FUNCTION_BLOCK Test_TimestampAsFilenameString EXTENDS TUnitTestBase
VAR
END_VAR

METHOD  Execute
VAR_INST
    TimeStruct : TIMESTRUCT := (wDay := 23, wMonth := 12, wYear := 1945, wHour := 22, wMinute := 20, wSecond := 18, wMilliseconds := 512);
END_VAR
Assertion.AssertEquals_STRING(
    Expected := '1945-12-23 22-20-18',
    Actual   := F_TimestampAsFilenameString(TimeStruct),
    ObjectName := _TestName,
    VariableName  := 'F_TimeAsString_ms(TimeStruct)');


Test_Finished();
END_METHOD

END_FUNCTION_BLOCK

(* stored: Version 1.1.0.1, ProductVersion 3.1.4024.3
   POU Test_TimestampAsFilenameString: Id {64d9bd98-83a2-4f8f-adab-051bd61aeff4}, SpecialFunc None
   Method Execute: Id {8659a975-d705-44ea-8d38-55144e853533} *)
